Yaskawa INFORM job: TEST-22R2.JBI

/JOB
//NAME TEST-22R2
///FOLDERNAME INNE
//POS
///NPOS 1,1,0,0,0,0
///TOOL 0
///POSTYPE PULSE
///PULSE
C00000=104062,-22335,-18949,19277,77654,53827
BC00000=44424,188252,600210
//INST
///DATE 2023/11/01 18:40
///ATTR SC,RW
///GROUP1 RB1,BS1
NOP
'test-22r2
MOVJ C00000 BC00000 VJ=100.00
END
